TYPE stCu_Header : 
STRUCT
    {attribute addProperty Name "<#Next on Passed#>"}
    NextOnPassed : enumStations;
    {attribute addProperty Name "<#Next on Failed#>"}
    NextOnFailed : enumStations;
END_STRUCT
END_TYPE

(* stored: Version 1.1.0.1, ProductVersion 3.1.4024.6
   DUT stCu_Header: Id {f7f4a5a4-14f1-4feb-be79-cb8509d968ec} *)
